FUNCTION_BLOCK DataMux
  (* Version 1.0, 2007-08-28, Goran Cengic, Chalmers *)
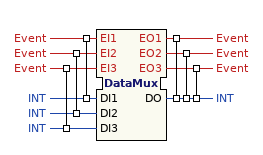
  EVENT_INPUT
    EI1 WITH DI1;
    EI2 WITH DI2;
    EI3 WITH DI3;
  END_EVENT
  EVENT_OUTPUT
    EO1 WITH DO;
    EO2 WITH DO;
    EO3 WITH DO;
  END_EVENT
  VAR_INPUT
    DI1 : INT;
    DI2 : INT;
    DI3 : INT;
  END_VAR
  VAR_OUTPUT
    DO : INT;
  END_VAR
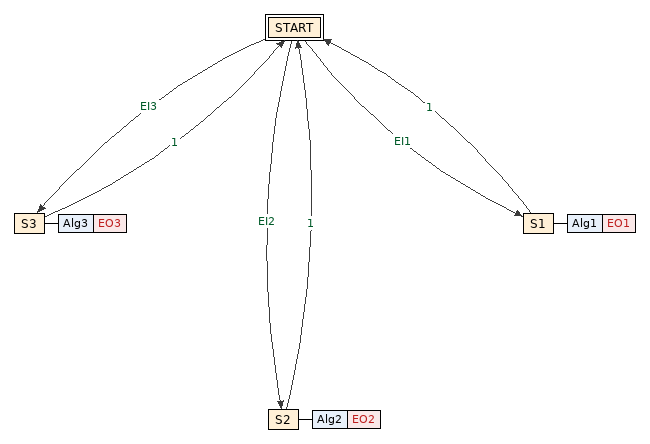
  EC_STATES
    START;
    S1 : Alg1 -> EO1;
    S2 : Alg2 -> EO2;
    S3 : Alg3 -> EO3;
  END_STATES
  EC_TRANSITIONS
    START TO S1 := EI1;
    S1 TO START := 1;
    START TO S2 := EI2;
    S2 TO START := 1;
    START TO S3 := EI3;
    S3 TO START := 1;
  END_TRANSITIONS
  ALGORITHM Alg1 IN Java:
DO = DI1;
  END_ALGORITHM
  ALGORITHM Alg2 IN Java:
DO = DI2;
  END_ALGORITHM
  ALGORITHM Alg3 IN Java:
DO = DI3;
  END_ALGORITHM
END_FUNCTION_BLOCK
